// Two different mistakes with two different answers. Folding them together would
// send the reader to the wrong argument: an empty label is usually a missing
// string, a null test a missing instance.
FUNCTION_BLOCK TEST_RegistryRejectsEmptyLabelAndNullTest IMPLEMENTS I_Test
VAR
	Registry  : TestRegistry<4>;
	Fake	  : FakeTest;
	NoTestRef : I_Test;
	Budgets	  : ST_TestBudgets;

	ExpectedFault : E_RegistrationFault;
	ActualFault	  : E_RegistrationFault;
	ExpectedCount : UDINT;
	ActualCount	  : UDINT;
END_VAR

METHOD Run : BOOL
VAR_INPUT
	Enable : BOOL;
	Test   : I_TestAssertions;
END_VAR
ActualFault	  := Registry.TryClaim(Fake, '', Budgets);
ExpectedFault := E_RegistrationFault.EmptyLabel;
Test.AssertEqual(ExpectedFault, ActualFault, 'empty label refused');

ActualFault	  := Registry.TryClaim(NoTestRef, 'Has a label but no test', Budgets);
ExpectedFault := E_RegistrationFault.NoTest;
Test.AssertEqual(ExpectedFault, ActualFault, 'null test refused as NoTest');

ExpectedCount := 0;
ActualCount	  := Registry.Count;
Test.AssertEqual(ExpectedCount, ActualCount, 'neither took a slot');

Run := TRUE;
END_METHOD

END_FUNCTION_BLOCK

(* stored: Version 1.1.0.1, ProductVersion 3.1.4026.18
   POU TEST_RegistryRejectsEmptyLabelAndNullTest: Id {327a8414-466d-4d07-b3bf-13355d587e73}, SpecialFunc None
   Folder I_Test: Id {25f15ece-8423-444a-8fec-0b98d1b372e3}
   Method Run: Id {a6cf22c3-38c4-415f-a71b-b45154e1ffac} *)
